# EPICS substitutions: Db/superv-freia.substitutions
file "diskTable.template" { pattern
{P,  DEV,  PASSWD, CHAN}
{"test-vm2", "disk", "freia_secret", 1}
}
